TYPE RxRemote :
STRUCT
	udp_key 	: DINT;
	comau 		: ControlComau;
END_STRUCT
END_TYPE

(* stored: Version 1.1.0.1, ProductVersion 3.1.4020.12
   DUT RxRemote: Id {7c5e24ba-f7d3-4959-970d-30aad538bc77} *)
